Fanuc TP program (LS listing): BOTTOM.LS

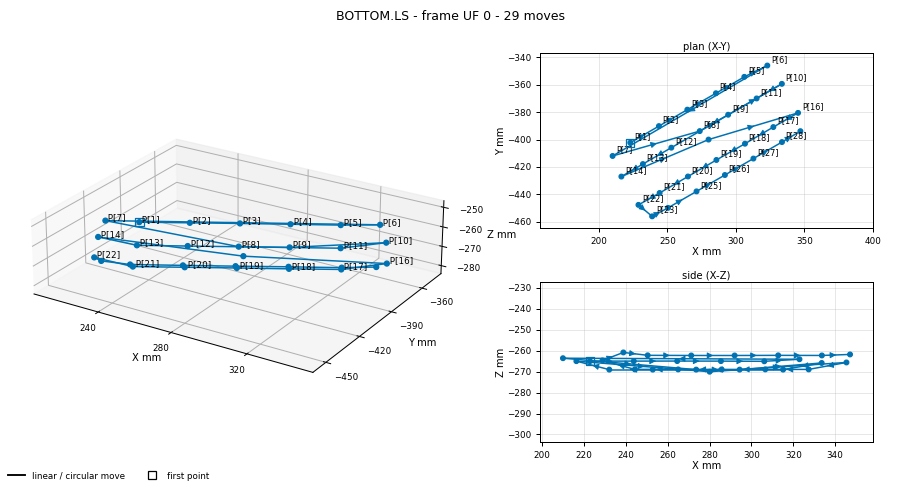
[picture p0: tool path of BOTTOM.LS in frame UF 0, 29 of 29 moves have a stored position in this frame; points joined in program order, loops and branches not executed]
/PROG  BOTTOM.LS
/ATTR
OWNER       = MNEDITOR;
COMMENT     = "";
PROG_SIZE   = 636;
CREATE      = DATE 23-01-07  TIME 11:59:14;
MODIFIED    = DATE 23-01-07  TIME 12:02:18;
FILE_NAME   = ;
VERSION     = 0;
LINE_COUNT  = 4;
MEMORY_SIZE = 992;
PROTECT     = READ_WRITE;
TCD:  STACK_SIZE	= 0,
      TASK_PRIORITY	= 50,
      TIME_SLICE	= 0,
      BUSY_LAMP_OFF	= 0,
      ABORT_REQUEST	= 0,
      PAUSE_REQUEST	= 0;
DEFAULT_GROUP	= 1,*,*,*,*;
CONTROL_CODE	= 00000000 00000000;
/MN
   1:J P[1] 100% FINE    ;
   2:L P[2] 100mm/sec CNT0    ;
   3:L P[3] 100mm/sec CNT0    ;
   4:L P[4] 100mm/sec CNT0    ;
   5:L P[5] 100mm/sec CNT0    ;
   6:L P[6] 100mm/sec CNT0    ;
   7:L P[7] 100mm/sec CNT0    ;
   8:L P[8] 100mm/sec CNT0    ;
   9:L P[9] 100mm/sec CNT0    ;
   10:L P[10] 100mm/sec CNT0    ;
   11:L P[11] 100mm/sec CNT0    ;
   12:L P[12] 100mm/sec CNT0    ;
   13:L P[13] 100mm/sec CNT0    ;
   14:L P[14] 100mm/sec CNT0    ;
   15:L P[15] 100mm/sec CNT0    ;
   16:L P[16] 100mm/sec CNT0    ;
   17:L P[17] 100mm/sec CNT0    ;
   18:L P[18] 100mm/sec CNT0    ;
   19:L P[19] 100mm/sec CNT0    ;
   20:L P[20] 100mm/sec CNT0    ;
   21:L P[21] 100mm/sec CNT0    ;
   22:L P[22] 100mm/sec CNT0    ;
   23:L P[23] 100mm/sec CNT0    ;
   24:L P[24] 100mm/sec CNT0    ;
   25:L P[25] 100mm/sec CNT0    ;
   26:L P[26] 100mm/sec CNT0    ;
   27:L P[27] 100mm/sec CNT0    ;
   28:L P[28] 100mm/sec CNT0    ;
   29:L P[29] 100mm/sec CNT0    ;
/POS
P[1]{
   GP1:
	UF : 0, UT : 6,		CONFIG : 'N U T, 0, 0, 0',
	X =  222.838  mm,	Y =   -402.264  mm,	Z =   -264.942  mm,
	W =  90.000 deg,	P =   0.000 deg,	R =   90.000 deg
};
P[2]{
   GP1:
	UF : 0, UT : 6,		CONFIG : 'N U T, 0, 0, 0',
	X =  243.762  mm,	Y =   -390.158  mm,	Z =   -264.940  mm,
	W =  90.000 deg,	P =   0.000 deg,	R =   90.000 deg
};
P[3]{
   GP1:
	UF : 0, UT : 6,		CONFIG : 'N U T, 0, 0, 0',
	X =  264.501  mm,	Y =   -378.148  mm,	Z =   -264.921  mm,
	W =  90.000 deg,	P =   0.000 deg,	R =   90.000 deg
};
P[4]{
   GP1:
	UF : 0, UT : 6,		CONFIG : 'N U T, 0, 0, 0',
	X =  285.398  mm,	Y =   -366.158  mm,	Z =   -264.948  mm,
	W =  90.000 deg,	P =   0.000 deg,	R =   90.000 deg
};
P[5]{
   GP1:
	UF : 0, UT : 6,		CONFIG : 'N U T, 0, 0, 0',
	X =  306.123  mm,	Y =   -354.184  mm,	Z =   -265.035  mm,
	W =  90.000 deg,	P =   0.000 deg,	R =   90.000 deg
};
P[6]{
   GP1:
	UF : 0, UT : 6,		CONFIG : 'N U T, 0, 0, 0',
	X =  322.922  mm,	Y =   -345.918  mm,	Z =   -264.055  mm,
	W =  90.000 deg,	P =   0.000 deg,	R =   90.000 deg
};
P[7]{
   GP1:
	UF : 0, UT : 6,		CONFIG : 'N U T, 0, 0, 0',
	X =  209.929  mm,	Y =   -411.968  mm,	Z =   -263.553  mm,
	W =  90.000 deg,	P =   0.000 deg,	R =   90.000 deg
};
P[8]{
   GP1:
	UF : 0, UT : 6,		CONFIG : 'N U T, 0, 0, 0',
	X =  273.567  mm,	Y =   -393.811  mm,	Z =   -269.000  mm,
	W =  90.000 deg,	P =   0.000 deg,	R =   90.000 deg
};
P[9]{
   GP1:
	UF : 0, UT : 6,		CONFIG : 'N U T, 0, 0, 0',
	X =  294.327  mm,	Y =   -381.866  mm,	Z =   -269.000  mm,
	W =  90.000 deg,	P =   0.000 deg,	R =   90.000 deg
};
P[10]{
   GP1:
	UF : 0, UT : 6,		CONFIG : 'N U T, 0, 0, 0',
	X =  333.546  mm,	Y =   -359.291  mm,	Z =   -265.831  mm,
	W =  90.000 deg,	P =   0.000 deg,	R =   90.000 deg
};
P[11]{
   GP1:
	UF : 0, UT : 6,		CONFIG : 'N U T, 0, 0, 0',
	X =  315.101  mm,	Y =   -369.964  mm,	Z =   -269.000  mm,
	W =  90.000 deg,	P =   0.000 deg,	R =   90.000 deg
};
P[12]{
   GP1:
	UF : 0, UT : 6,		CONFIG : 'N U T, 0, 0, 0',
	X =  252.827  mm,	Y =   -405.913  mm,	Z =   -269.000  mm,
	W =  90.000 deg,	P =   0.000 deg,	R =   90.000 deg
};
P[13]{
   GP1:
	UF : 0, UT : 6,		CONFIG : 'N U T, 0, 0, 0',
	X =  232.061  mm,	Y =   -417.877  mm,	Z =   -269.000  mm,
	W =  90.000 deg,	P =   0.000 deg,	R =   90.000 deg
};
P[14]{
   GP1:
	UF : 0, UT : 6,		CONFIG : 'N U T, 0, 0, 0',
	X =  216.334  mm,	Y =   -427.017  mm,	Z =   -264.956  mm,
	W =  90.000 deg,	P =   0.000 deg,	R =   90.000 deg
};
P[15]{
   GP1:
	UF : 0, UT : 6,		CONFIG : 'N U T, 0, 0, 0',
	X =  280.000  mm,	Y =   -400.000  mm,	Z =   -270.000  mm,
	W =  90.000 deg,	P =   0.000 deg,	R =   90.000 deg
};
P[16]{
   GP1:
	UF : 0, UT : 6,		CONFIG : 'N U T, 0, 0, 0',
	X =  345.369  mm,	Y =   -380.490  mm,	Z =   -265.581  mm,
	W =  90.000 deg,	P =   0.000 deg,	R =   90.000 deg
};
P[17]{
   GP1:
	UF : 0, UT : 6,		CONFIG : 'N U T, 0, 0, 0',
	X =  327.315  mm,	Y =   -390.859  mm,	Z =   -268.904  mm,
	W =  90.000 deg,	P =   0.000 deg,	R =   90.000 deg
};
P[18]{
   GP1:
	UF : 0, UT : 6,		CONFIG : 'N U T, 0, 0, 0',
	X =  306.600  mm,	Y =   -403.019  mm,	Z =   -268.900  mm,
	W =  90.000 deg,	P =   0.000 deg,	R =   90.000 deg
};
P[19]{
   GP1:
	UF : 0, UT : 6,		CONFIG : 'N U T, 0, 0, 0',
	X =  285.734  mm,	Y =   -414.898  mm,	Z =   -268.907  mm,
	W =  90.000 deg,	P =   0.000 deg,	R =   90.000 deg
};
P[20]{
   GP1:
	UF : 0, UT : 6,		CONFIG : 'N U T, 0, 0, 0',
	X =  264.965  mm,	Y =   -426.965  mm,	Z =   -268.903  mm,
	W =  90.000 deg,	P =   0.000 deg,	R =   90.000 deg
};
P[21]{
   GP1:
	UF : 0, UT : 6,		CONFIG : 'N U T, 0, 0, 0',
	X =  244.275  mm,	Y =   -439.001  mm,	Z =   -268.898  mm,
	W =  90.000 deg,	P =   0.000 deg,	R =   90.000 deg
};
P[22]{
   GP1:
	UF : 0, UT : 6,		CONFIG : 'N U T, 0, 0, 0',
	X =  228.805  mm,	Y =   -447.692  mm,	Z =   -264.629  mm,
	W =  90.000 deg,	P =   0.000 deg,	R =   90.000 deg
};
P[23]{
   GP1:
	UF : 0, UT : 6,		CONFIG : 'N U T, 0, 0, 0',
	X =  238.794  mm,	Y =   -456.075  mm,	Z =   -260.799  mm,
	W =  90.000 deg,	P =   0.000 deg,	R =   90.000 deg
};
P[24]{
   GP1:
	UF : 0, UT : 6,		CONFIG : 'N U T, 0, 0, 0',
	X =  250.398  mm,	Y =   -449.864  mm,	Z =   -262.177  mm,
	W =  90.000 deg,	P =   0.000 deg,	R =   90.000 deg
};
P[25]{
   GP1:
	UF : 0, UT : 6,		CONFIG : 'N U T, 0, 0, 0',
	X =  271.222  mm,	Y =   -437.838  mm,	Z =   -262.248  mm,
	W =  90.000 deg,	P =   0.000 deg,	R =   90.000 deg
};
P[26]{
   GP1:
	UF : 0, UT : 6,		CONFIG : 'N U T, 0, 0, 0',
	X =  291.934  mm,	Y =   -425.882  mm,	Z =   -262.254  mm,
	W =  90.000 deg,	P =   0.000 deg,	R =   90.000 deg
};
P[27]{
   GP1:
	UF : 0, UT : 6,		CONFIG : 'N U T, 0, 0, 0',
	X =  312.762  mm,	Y =   -413.861  mm,	Z =   -262.190  mm,
	W =  90.000 deg,	P =   0.000 deg,	R =   90.000 deg
};
P[28]{
   GP1:
	UF : 0, UT : 6,		CONFIG : 'N U T, 0, 0, 0',
	X =  333.625  mm,	Y =   -401.813  mm,	Z =   -262.238  mm,
	W =  90.000 deg,	P =   0.000 deg,	R =   90.000 deg
};
P[29]{
   GP1:
	UF : 0, UT : 6,		CONFIG : 'N U T, 0, 0, 0',
	X =  347.080  mm,	Y =   -393.870  mm,	Z =   -261.753  mm,
	W =  90.000 deg,	P =   0.000 deg,	R =   90.000 deg
};
/END
